// TIA Portal project "prova2" (V15.1)

(* hardware
DEVICE "S7-1200 station_1"  S7-1200 Station
   slot 0: "Telaio di montaggio_0"  S7-1200 Rack  Rack  V1.0
   slot 1: "PLC_1"  CPU 1214C DC/DC/DC  6ES7 214-1AG40-0XB0  V4.2
*)

// ===== PLC "PLC_1"  CPU 1214C DC/DC/DC =====

DATA_BLOCK "Blocco_dati"   // DB1
{ S7_Optimized_Access := 'TRUE' }
VERSION : 0.1
   VAR RETAIN
      "array" : Array[0..9] of Int;
      contatore : Int;
   END_VAR
BEGIN
END_DATA_BLOCK

ORGANIZATION_BLOCK "Main"   // OB1, LAD, ProgramCycle
TITLE = "Main Program Sweep (Cycle)"
{ S7_Optimized_Access := 'TRUE' }
VERSION : 0.1
   VAR_INPUT
      Initial_Call : Bool;   // Initial call of this OB
      Remanence : Bool;   // =True, if remanent data are available
   END_VAR
BEGIN
END_ORGANIZATION_BLOCK

ORGANIZATION_BLOCK "Cyclic interrupt"   // OB30, LAD, CyclicInterrupt
{ S7_Optimized_Access := 'TRUE' }
VERSION : 0.1
   VAR_INPUT
      Initial_Call : Bool;   // Initial call of this OB
      Event_Count : Int;   // Events discarded
   END_VAR
BEGIN

REGION Network 1
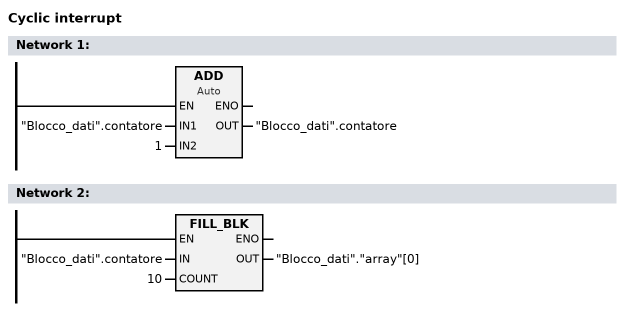
   RUNG wire#powerrail
      Add(in1 := "Blocco_dati".contatore, in2 := 1, out => "Blocco_dati".contatore)
   END_RUNG
   // the same network as SCL:
   "Blocco_dati".contatore := "Blocco_dati".contatore + 1;
END_REGION

REGION Network 2
   RUNG wire#powerrail
      FillBlockI(in := "Blocco_dati".contatore, count := 10, out => "Blocco_dati"."array"[0])
   END_RUNG
   // the same network as SCL:
   FILL_BLK(IN := "Blocco_dati".contatore, COUNT := 10, OUT => "Blocco_dati"."array"[0]);
END_REGION
END_ORGANIZATION_BLOCK